// Mitsubishi GX Works2 project: 123   PLC: FX0S/FX0

PROGRAM MAIN
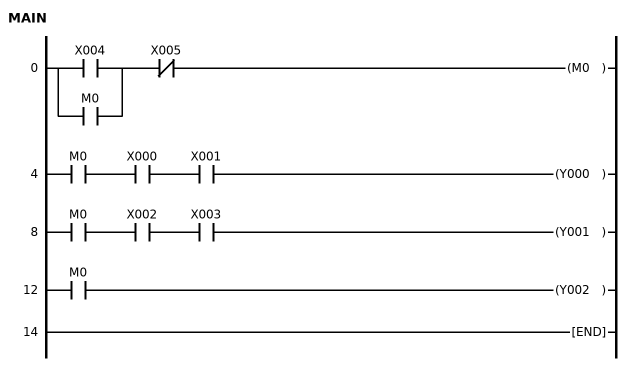
0     LD      X004
      OR      M0
      ANI     X005
      OUT     M0
4     LD      M0
      AND     X000
      AND     X001
      OUT     Y000
8     LD      M0
      AND     X002
      AND     X003
      OUT     Y001
12    LD      M0
      OUT     Y002
14    END
END_PROGRAM
